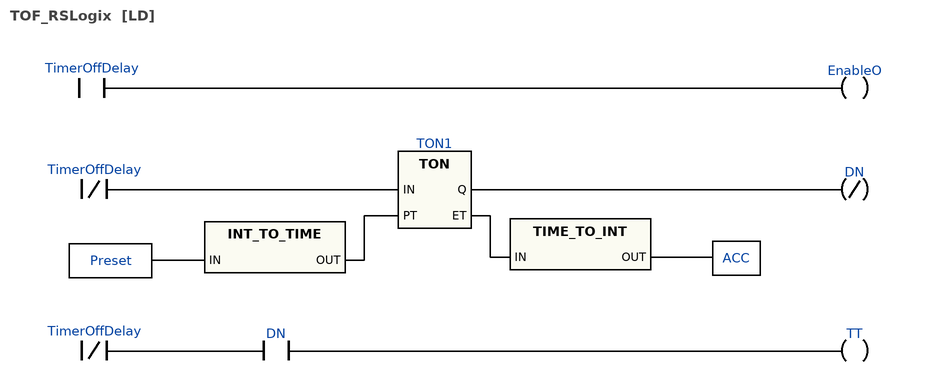
(* LD diagram, written out as Structured Text *)
EnableO := TimerOffDelay;
TON1(IN := NOT TimerOffDelay, PT := INT_TO_TIME(Preset));
DN := NOT TON1.Q;
ACC := TIME_TO_INT(TON1.ET);
TT := NOT TimerOffDelay AND DN;
END_FUNCTION_BLOCK

FUNCTION_BLOCK TON_RSLogix
  VAR_INPUT
    TimerOnDelay : BOOL := FALSE;
    Preset : INT := 0;
  END_VAR
  VAR_OUTPUT
    EnableO : BOOL := FALSE;
    DN : BOOL := FALSE;
    ACC : INT := 0;
    TT : BOOL := FALSE;
  END_VAR
  VAR
    TON1 : TON;
  END_VAR

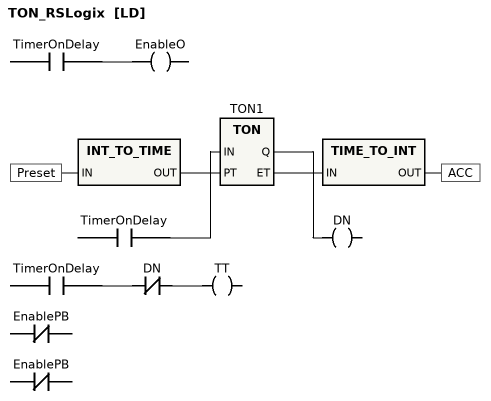
(* LD diagram, written out as Structured Text *)
EnableO := TimerOnDelay;
TON1(IN := TimerOnDelay, PT := INT_TO_TIME(Preset));
DN := TON1.Q;
ACC := TIME_TO_INT(TON1.ET);
TT := TimerOnDelay AND NOT DN;
(* drawn but not wired to any output: EnablePB, EnablePB *)
END_FUNCTION_BLOCK

FUNCTION_BLOCK HMI_Safety
  VAR_IN_OUT
    ESTOP_FP : BOOL := FALSE;
    CommOK : BOOL := FALSE;
  END_VAR
  VAR_INPUT
    FirstScanOneShot : BOOL;
    NoEStopCHA : BOOL;
    NoEStopCHB : BOOL;
  END_VAR
  VAR_OUTPUT
    ESTOP_FaultReset : BOOL := FALSE;
    ESTOP_O1 : BOOL := FALSE;
    NoEstop : BOOL := FALSE;
  END_VAR
  VAR_INPUT
    AutoModeS : BOOL;
    ManModeS : BOOL;
  END_VAR
  VAR_IN_OUT
    AutoMan_FP : BOOL := FALSE;
  END_VAR
  VAR_OUTPUT
    AutoMan_FaultReset : BOOL := FALSE;
    AutoManDebounce_PRE : INT := 200;
    AutoManDebounce_TT : BOOL := FALSE;
  END_VAR
  VAR_IN_OUT
    Pos1Int : BOOL := FALSE;
    Pos2Int : BOOL := FALSE;
  END_VAR
  VAR_OUTPUT
    AutoMan_O1 : BOOL := FALSE;
    AutoMan_O2 : BOOL := FALSE;
    AutoMode : BOOL := FALSE;
    ManualMode : BOOL := FALSE;
  END_VAR
  VAR_IN_OUT
    PendantOK_FP : BOOL := FALSE;
  END_VAR
  VAR_OUTPUT
    PendantOK_FaultReset : BOOL := FALSE;
  END_VAR
  VAR_INPUT
    E130CREP : BOOL;
    E134CREP : BOOL;
    HMI_Select : BOOL;
  END_VAR
  VAR_IN_OUT
    Selected : BOOL := FALSE;
  END_VAR
  VAR_INPUT
    HMI_SelectionOK : BOOL;
    Gates_SelectAvail : BOOL;
    EnablePB : BOOL;
  END_VAR
  VAR_IN_OUT
    Enable : BOOL := FALSE;
    PHMIEnable : BOOL := FALSE;
    EnableAntiRepeat : BOOL := FALSE;
  END_VAR
  VAR_OUTPUT
    EnableTmr_PRE : INT := 600;
    EnableTmr_DN : BOOL := FALSE;
  END_VAR
  VAR_INPUT
    OneHMIEnabled : BOOL;
    Gates_OneRobotToolMinorReq : BOOL;
    OneHMIMode : BOOL;
  END_VAR
  VAR_OUTPUT
    PendEnable : BOOL := FALSE;
    PendOk : BOOL := FALSE;
  END_VAR
  VAR_INPUT
    AlwaysOff : BOOL;
    FltBcn : BOOL;
  END_VAR
  VAR_OUTPUT
    O_FaultLT : BOOL := FALSE;
  END_VAR
  VAR_INPUT
    ResetLT : BOOL;
  END_VAR
  VAR_OUTPUT
    O_ResetLT : BOOL := FALSE;
  END_VAR
  VAR_INPUT
    AutoInitLT : BOOL;
  END_VAR
  VAR_OUTPUT
    O_AutoInitLT : BOOL := FALSE;
  END_VAR
  VAR_INPUT
    CombinedStatus : BOOL;
  END_VAR
  VAR_OUTPUT
    NoSafetyFaults : BOOL := FALSE;
  END_VAR
  VAR_IN_OUT
    BackCheck_NoEStop : BOOL := FALSE;
    BackCheck_NoSafetyFaults : BOOL := FALSE;
  END_VAR
  VAR
    ESTOP1 : ESTOP;
    TOF1 : TOF_RSLogix;
    FPMS1 : FPMS;
    ENPEN1 : ENPEN;
    TON1 : TON_RSLogix;
  END_VAR
  VAR  (* added by the conversion: wires and edge detectors of the diagram *)
    _MOV_E_Int30_ : ANY;
    _MOV_E_Int30_OUT : INT;
    _MOV_E_Int83_ : ANY;
    _MOV_E_Int83_OUT : INT;
  END_VAR

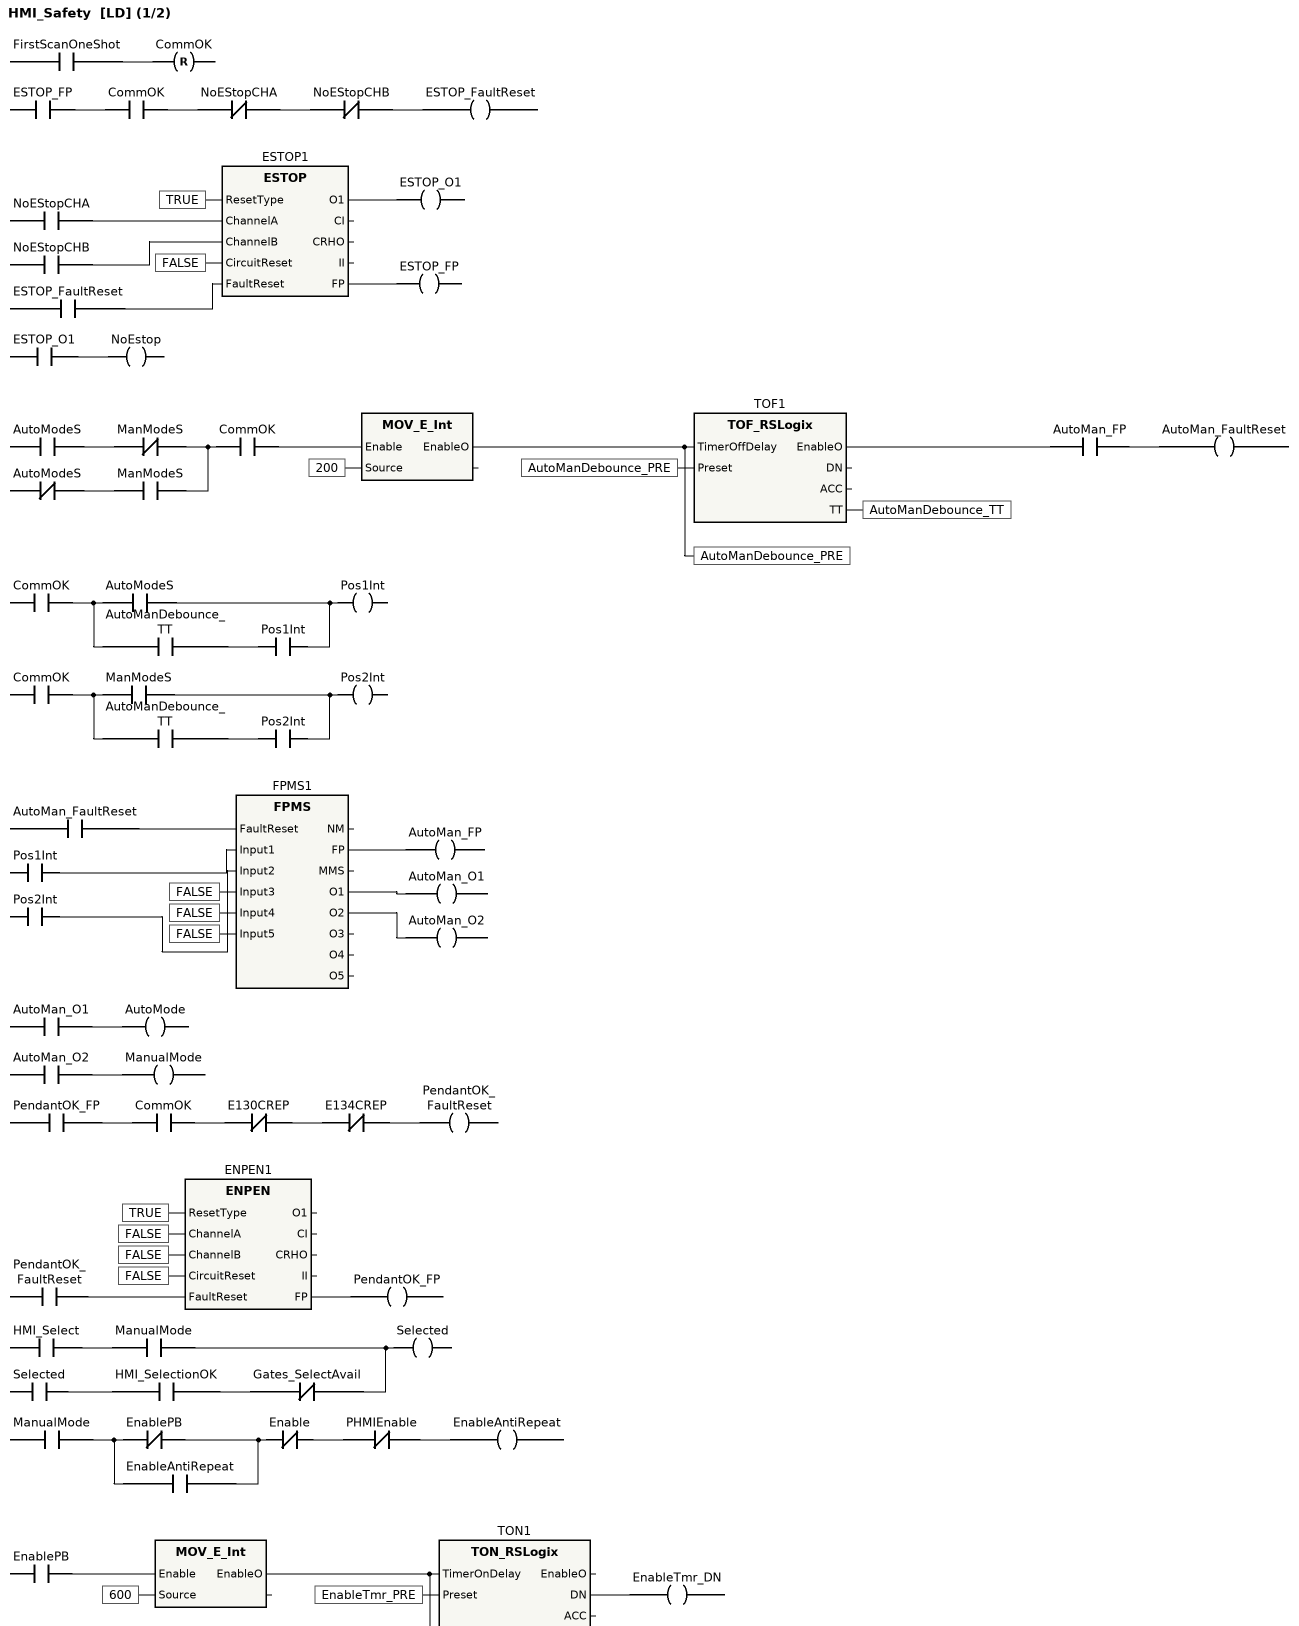
(* LD diagram, written out as Structured Text *)
IF FirstScanOneShot THEN CommOK := FALSE; END_IF;
ESTOP_FaultReset := ESTOP_FP AND CommOK AND NOT NoEStopCHA AND NOT NoEStopCHB;
ESTOP1(ResetType := TRUE, ChannelA := NoEStopCHA, ChannelB := NoEStopCHB, CircuitReset := FALSE, FaultReset := ESTOP_FaultReset);
ESTOP_O1 := ESTOP1.O1;
ESTOP_FP := ESTOP1.FP;
NoEstop := ESTOP_O1;
_MOV_E_Int30_OUT := MOV_E_Int(Enable := (AutoModeS AND NOT ManModeS OR NOT AutoModeS AND ManModeS) AND CommOK, Source := 200,  => _MOV_E_Int30_);
TOF1(TimerOffDelay := _MOV_E_Int30_OUT, Preset := AutoManDebounce_PRE);
AutoMan_FaultReset := TOF1.EnableO AND AutoMan_FP;
AutoManDebounce_PRE := _MOV_E_Int30_OUT;
AutoManDebounce_TT := TOF1.TT;
Pos1Int := CommOK AND (AutoModeS OR AutoManDebounce_TT AND Pos1Int);
Pos2Int := CommOK AND (ManModeS OR AutoManDebounce_TT AND Pos2Int);
FPMS1(FaultReset := AutoMan_FaultReset, Input1 := Pos1Int, Input2 := Pos2Int, Input3 := FALSE, Input4 := FALSE, Input5 := FALSE);
AutoMan_FP := FPMS1.FP;
AutoMan_O1 := FPMS1.O1;
AutoMan_O2 := FPMS1.O2;
AutoMode := AutoMan_O1;
ManualMode := AutoMan_O2;
PendantOK_FaultReset := PendantOK_FP AND CommOK AND NOT E130CREP AND NOT E134CREP;
ENPEN1(ResetType := TRUE, ChannelA := FALSE, ChannelB := FALSE, CircuitReset := FALSE, FaultReset := PendantOK_FaultReset);
PendantOK_FP := ENPEN1.FP;
Selected := HMI_Select AND ManualMode OR Selected AND HMI_SelectionOK AND NOT Gates_SelectAvail;
EnableAntiRepeat := ManualMode AND (NOT EnablePB OR EnableAntiRepeat) AND NOT Enable AND NOT PHMIEnable;
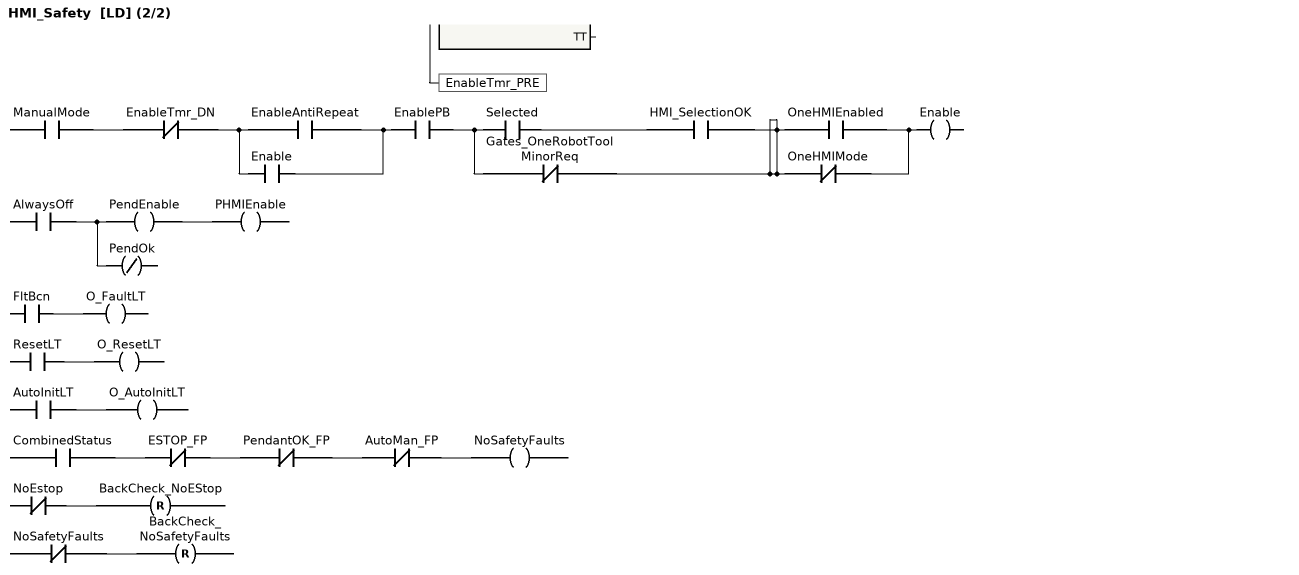
_MOV_E_Int83_OUT := MOV_E_Int(Enable := EnablePB, Source := 600,  => _MOV_E_Int83_);
EnableTmr_PRE := _MOV_E_Int83_OUT;
TON1(TimerOnDelay := _MOV_E_Int83_OUT, Preset := EnableTmr_PRE);
EnableTmr_DN := TON1.DN;
Enable := ManualMode AND NOT EnableTmr_DN AND (EnableAntiRepeat OR Enable) AND EnablePB AND ((NOT Gates_OneRobotToolMinorReq OR Selected AND HMI_SelectionOK) AND OneHMIEnabled OR (Selected AND HMI_SelectionOK OR NOT Gates_OneRobotToolMinorReq) AND NOT OneHMIMode);
PendEnable := AlwaysOff;
PHMIEnable := AlwaysOff;
PendOk := NOT AlwaysOff;
O_FaultLT := FltBcn;
O_ResetLT := ResetLT;
O_AutoInitLT := AutoInitLT;
NoSafetyFaults := CombinedStatus AND NOT ESTOP_FP AND NOT PendantOK_FP AND NOT AutoMan_FP;
IF NOT NoEstop THEN BackCheck_NoEStop := FALSE; END_IF;
IF NOT NoSafetyFaults THEN BackCheck_NoSafetyFaults := FALSE; END_IF;
END_FUNCTION_BLOCK

FUNCTION_BLOCK Emergency_Stop
  VAR_IN_OUT
    EStop_FP : BOOL := FALSE;
  END_VAR
  VAR_INPUT
    CommOK : BOOL;
    NoEStopCHA : BOOL;
    NoEStopCHB : BOOL;
  END_VAR
  VAR_OUTPUT
    EStop_FaultReset : BOOL;
    EStop_O1 : BOOL;
    NoEstop : BOOL;
  END_VAR
  VAR_INPUT
    AutoModeS : BOOL;
    ManModeS : BOOL;
  END_VAR
  VAR_IN_OUT
    AutoMan_FP : BOOL;
  END_VAR
  VAR_OUTPUT
    AutoMan_FaultReset : BOOL;
    AutoManDebounce_PRE : BOOL;
    AutoManDebounce_TT : BOOL;
  END_VAR
  VAR_IN_OUT
    Pos1Int : BOOL;
    Pos2Int : BOOL;
  END_VAR
  VAR_OUTPUT
    AutoMan_O1 : BOOL;
    AutoMan_O2 : BOOL;
    AutoMode : BOOL;
    ManualMode : BOOL;
  END_VAR
  VAR_IN_OUT
    PendantOK_FP : BOOL;
  END_VAR
  VAR_OUTPUT
    PendantOK_FaultReset : BOOL;
  END_VAR
  VAR_INPUT
    E130CREP : BOOL;
    E134CREP : BOOL;
    HMI_Select : BOOL;
  END_VAR
  VAR_IN_OUT
    Selected : BOOL;
  END_VAR
  VAR_INPUT
    HMI_SelectionOK : BOOL;
    Gates_SelectAvail : BOOL;
    EnablePB : BOOL;
  END_VAR
  VAR_IN_OUT
    Enable : BOOL;
    PHMIEnable : BOOL;
    EnableAntiRepeat : BOOL;
  END_VAR
  VAR_OUTPUT
    EnableTmr_PRE : BOOL;
    EnableTmr_EN : BOOL;
    EnableTmr_DN : BOOL;
  END_VAR
  VAR_INPUT
    OneHMIEnabled : BOOL;
    Gates_OneRobotToolMinorReq : BOOL;
    OneHMIMode : BOOL;
  END_VAR
  VAR_OUTPUT
    PendEnable : BOOL;
    PendOk : BOOL;
    RungComment : BOOL;
  END_VAR
  VAR_INPUT
    AlwaysOff : BOOL;
    FltBcn : BOOL;
  END_VAR
  VAR_OUTPUT
    O_FaultLT : BOOL;
  END_VAR
  VAR_INPUT
    ResetLT : BOOL;
  END_VAR
  VAR_OUTPUT
    O_ResetLT : BOOL;
  END_VAR
  VAR_INPUT
    AutoInitLT : BOOL;
  END_VAR
  VAR_OUTPUT
    O_AutoInitLT : BOOL;
  END_VAR
  VAR_INPUT
    CombinedStatus : BOOL;
  END_VAR
  VAR_OUTPUT
    NoSafetyFaults : BOOL;
  END_VAR
  VAR_IN_OUT
    BackCheck_NoEStop : BOOL;
    BackCheck_NoSafetyFaults : BOOL;
  END_VAR

(* LD diagram, written out as Structured Text *)
END_FUNCTION_BLOCK

FUNCTION_BLOCK HMI_Safety_FullAlgorithm
  VAR
    ESTOP_FP : BOOL := FALSE;
  END_VAR
  VAR_IN_OUT
    CommOK : BOOL;
  END_VAR
  VAR_INPUT
    FirstScanOneShot : BOOL;
    NoEStopCHA : BOOL;
    NoEStopCHB : BOOL;
  END_VAR
  VAR
    ESTOP_FaultReset : BOOL;
    ESTOP_O1 : BOOL;
  END_VAR
  VAR_OUTPUT
    NoEstop : BOOL;
  END_VAR
  VAR_INPUT
    AutoModeS : BOOL;
    ManModeS : BOOL;
  END_VAR
  VAR
    AutoMan_FP : BOOL;
    AutoMan_FaultReset : BOOL;
    AutoManDebounce_PRE : BOOL;
    AutoManDebounce_TT : BOOL;
    Pos1Int : BOOL;
    Pos2Int : BOOL;
    AutoMan_O1 : BOOL;
    AutoMan_O2 : BOOL;
  END_VAR
  VAR_OUTPUT
    AutoMode : BOOL;
    ManualMode : BOOL;
  END_VAR
  VAR
    PendantOK_FP : BOOL;
    PendantOK_FaultReset : BOOL;
  END_VAR
  VAR_INPUT
    E130CREP : BOOL;
    E134CREP : BOOL;
    HMI_Select : BOOL;
  END_VAR
  VAR_OUTPUT
    Selected : BOOL;
  END_VAR
  VAR_INPUT
    HMI_SelectionOK : BOOL;
    Gates_SelectAvail : BOOL;
    EnablePB : BOOL;
  END_VAR
  VAR
    Enable : BOOL;
    PHMIEnable : BOOL;
    EnableAntiRepeat : BOOL;
    EnableTmr_PRE : BOOL;
  END_VAR
  VAR_OUTPUT
    EnableTmr_EN : BOOL;
  END_VAR
  VAR
    EnableTmr_DN : BOOL;
  END_VAR
  VAR_INPUT
    OneHMIEnabled : BOOL;
  END_VAR
  VAR
    Gates_OneRobotToolMinorReq : BOOL;
  END_VAR
  VAR_INPUT
    OneHMIMode : BOOL;
  END_VAR
  VAR_OUTPUT
    PendEnable : BOOL;
    PendOk : BOOL;
  END_VAR

(* LD diagram, written out as Structured Text *)
END_FUNCTION_BLOCK

FUNCTION MOV_E_Time : TIME
  VAR_INPUT
    Enable : BOOL;
    Source : TIME;
  END_VAR
  VAR_OUTPUT
    EnableO : BOOL;
  END_VAR

(* LD diagram, written out as Structured Text *)
END_FUNCTION

CONFIGURATION ExampleCell
END_CONFIGURATION
